FUNCTION_BLOCK FB_FormingBoardControl_V1
VAR_INPUT
    // ── Group / Interlocks ───────────────────────────────────────────────────────
    startGroup                   : BOOL;   // Start command (pulse / rising edge)
    stopGroup                    : BOOL;   // Stop command  (pressed / level)
    groupReset                   : BOOL;   // Group fault Reset (Comando reset falhas do grupo)

    // ── VFD per-drive status inputs ─────────────────────────────────────────────
    formingBoardTractionRollFault               : BOOL;   // VFD ready/healthy (master)
	formingBoardTractionRollCoolingFault  : BOOL;   // VFD ready/healthy (master)
    formingBoardTractionRollVfdRunFeedback         : BOOL;   // VFD RUN feedback  (master)
    formingBoardTractionRollVfdFaultFeedback       : BOOL;   // VFD fault         (master)
   
	formingBoardSuctionRollFault                : BOOL;   // VFD ready/healthy (slave)
	formingBoardSuctionRollCoolingFault		: BOOL;   // VFD ready/healthy (slave)	
	
    formingBoardSuctionVfdRunFeedback          : BOOL;   // VFD RUN feedback  (slave)
    formingBoardSuctionVfdFaultFeedback        : BOOL;   // VFD fault         (slave)

    // ── Speed Setpoints ─────────────────────────────────────────────────────────
    groupAutoSpeedMPM            : REAL;   // Auto speed setpoint [m/min]
    groupMaxSpeed                : REAL := 600.0; // Max allowed line speed [m/min]

    // ── Auto / Manual ───────────────────────────────────────────────────────────
    groupSpeedAutoMan            : BOOL;   // 0=Manual / 1=Auto
    groupManualSpeedMPM          : REAL := 50.0;  // Manual speed [m/min]

    // ── Feedbacks ───────────────────────────────────────────────────────────────
    masterTorqueFeedback         : REAL;   // [% or Nm]
    slaveTorqueFeedback          : REAL;   // [% or Nm]
    masterSpeedFeedback          : REAL;   // [m/min or %] — be consistent
    slaveSpeedFeedback           : REAL;   // [m/min or %] — be consistent

    // ── Ratio & Offsets ─────────────────────────────────────────────────────────
    masterSlaveGearRatio		: REAL := 1.0;   // Slave/Master speed ratio
// 	interGroupGearRatio			: REAL := 1.0;   // Speed diference btween groups
	
    slaveTorqueOfsset            : REAL := 0.0;   // (typo kept) torque trim [%/Nm]
    slaveSpeedOffset             : REAL := 10;    // Offset as % of master speed (+5 => +5%)

    // ── Torque control parameters ───────────────────────────────────────────────
    torqueLimitMinPct            : REAL := 5.0;   // Min torque [%]  (allow negative if regen)
    torqueLimitMaxPct            : REAL := 100.0; // Max torque [%]
    torqueDeadbandPct            : REAL := 1.0;   // |torque| below => 0 (noise cleanup)
	
    torqueFilterTime             : TIME := T#1MS;
    displayFilterTime             : TIME := T#20MS;	

    // ── Dynamics (for ramp block) ───────────────────────────────────────────────
    rampRate                     : REAL := 0.01;  // Ref accel mag in %/s (A_UP=+rampRate, A_DN=-rampRate)

    // ── Speed difference limit ──────────────────────────────────────────────────
    speedDiferenceLimit          : REAL := 5.0;
	
	
	
	
	//Headbox inputs
	
	//==============================================================
	// FORMING BOARD — WIRE EDGE OVERRUN SENSORS
	//==============================================================
	formingBoardWireOverrunOperatorSideSensor : BOOL;  // TRUE when wire overruns on operator side
	formingBoardWireOverrunDriveSideSensor    : BOOL;  // TRUE when wire overruns on drive/motor side	

	//==============================================================
	// HEADBOX LIPS OPENING CONTROL — VARIABLES
	//==============================================================
	
	// Position feedback and physical limits [mm]
	headboxLipsPositionFeedback_mm     : REAL;          // Actual lips opening [mm]
	headboxLipsMinOpening_mm           : REAL := 0.0;   // Minimum allowed opening [mm]
	headboxLipsMaxOpening_mm           : REAL := 25.0;  // Maximum allowed opening [mm]
	
	// Limit sensors (digital inputs)
	headboxLipsLimitFullyOpen          : BOOL;          // TRUE when fully open (max) limit sensor active
	headboxLipsLimitFullyClosed        : BOOL;          // TRUE when fully closed (min) limit sensor active
	
	// Manual jog commands (for manual mode)
	headboxLipsManualOpenCmd           : BOOL;          // Jog open while pressed
	headboxLipsManualCloseCmd          : BOOL;          // Jog close while pressed
	
	// Automatic positioning (for auto mode)
	headboxLipsTargetSetpoint_mm       : REAL;          // Desired lips opening [mm]
	headboxLipsAutoAdjustCmd           : BOOL;          // Pulse to start auto adjustment
	
		
	formingBoardRollUpCmd        : BOOL;  // Command to move forming board UP (active-high)
	formingBoardRollDownCmd      : BOOL;  // Command to move forming board DOWN (active-high)
	formingBoardRollLimitUpSensor    : BOOL;  // TRUE when upper limit is reached (prevents further UP)
	formingBoardRollLimitDownSensor  : BOOL;  // TRUE when lower limit is reached (prevents further DOWN)
	formingBoardRollUpDownMotorFault            : BOOL;  // TRUE = fault present → disables all movement	
	
	formingBoardStretchCmd           : BOOL;  // Jog command to stretch (increase tension)
	formingBoardUnstretchCmd         : BOOL;  // Jog command to unstretch (decrease tension)
	formingBoardLimitStretchSensor   : BOOL;  // TRUE when maximum stretch limit is reached
	formingBoardLimitUnstretchSensor : BOOL;  // TRUE when minimum stretch limit is reached
	formingBoardStretchMotorFault         : BOOL;  // Fault interlock for stretch unit
	
		
END_VAR

VAR_OUTPUT
    deviceState                  : STRING;
    groupFault                   : BOOL;   // Fault present (Falha do grupo)

    // ── Drive References (0..100%) ──────────────────────────────────────────────
    masterDriveSpeedRefPct       : REAL;   // Master reference [%]
    slaveDriveSpeedRefPct        : REAL;   // Slave  reference [%]
	nextGroupSpeedRefPct		 : REAL;   // Next group reference [%]
	nextGroupSpeedRefMPM		 : REAL;   // Next group reference [Meters per minute]
	
    // ── Torque limit to slave (from master torque path / or PID) ───────────────
    slaveDriveTorqueLimit        : REAL;   // [% or Nm]

    // ── Drive Commands ──────────────────────────────────────────────────────────
    masterDriveEnable            : BOOL;
    slaveDriveEnable             : BOOL;
    masterDriveReset             : BOOL;
    slaveDriveReset              : BOOL;

    // ── Diagnostics ─────────────────────────────────────────────────────────────
    currentSpeedDifence          : REAL;

    // ── Group status & HMI displays ────────────────────────────────────────────
    statusCode                   	: INT;    // 0=Idle, 1=Starting, 2=Running, 3=Fault (group)
	
    masterSpeedMPMFilteredDisplay   : REAL;   // Filtered master speed [m/min]
    slaveSpeedMPMFilteredDisplay    : REAL;   // Filtered slave  speed [m/min]
	
    masterTorqueFilteredDisplay  	: REAL;   // Master torque (raw)  [% or Nm]
    slaveTorqueFilteredDisplay   	: REAL;   // Slave torque (filtered) [% or Nm]

    // ── NEW: per-drive motor status codes ───────────────────────────────────────
    masterStatusCode             : INT;    // 0=Idle, 1=Starting, 2=Running, 3=Fault
    slaveStatusCode              : INT;    // 0=Idle, 1=Starting, 2=Running, 3=Fault
	
	//==============================================================
	// HEADBOX LIPS OPENING CONTROL — OUTPUTS
	//==============================================================
	
	// Drive outputs (modulated by PWM in automatic mode)
	headboxLipsOpenCmd                : BOOL;  // Output to open lips (PWM-modulated in Auto mode)
	headboxLipsCloseCmd               : BOOL;  // Output to close lips (PWM-modulated in Auto mode)
	headboxLipsPosition_mm       		  : REAL;  // Target − Feedback error [mm]
	
	//==============================================================
	// FORMING BOARD — ROLL DRIVE OUTPUTS
	//==============================================================
	formingBoardRollUp       : BOOL;  // Output to drive the forming board UP
	formingBoardRollDown     : BOOL;  // Output to drive the forming board DOWN
	
	//==============================================================
	// FORMING BOARD — STRETCH DRIVE OUTPUTS
	//==============================================================
	formingBoardStretch      : BOOL;  // Output to stretch (increase tension)
	formingBoardUnstretch    : BOOL;  // Output to unstretch (decrease tension)
		

	hmiAlarms 				: PaperMachine_TypeHmiAlarms; 	

END_VAR

VAR
    // ── Internals / Ramps ───────────────────────────────────────────────────────
    rampTargetPct                : REAL;   // 0..100% target into ramp
    instFB_Gen_SRamp             : FB_Gen_SRamp; // Your ramp FB

    // ── State & Edges ───────────────────────────────────────────────────────────
    state                        : INT;    // 0=IDLE,1=ENABLE,2=WAIT_EN,3=RAMP_EN,4=RUN,5=STOPPING,10=FAULT
    startGroupOld                : BOOL;
    stopGroupOld                 : BOOL;
    rStart                       : BOOL;
    rStop                        : BOOL;

    // ── Timers & thresholds ─────────────────────────────────────────────────────
    instTONEnableWait            : TON;
    instTONStopWait              : TON;
    enableTimeout                : TIME := T#5s;  // Wait for op-enable
    stopTimeout                  : TIME := T#8s;  // Max wait to speed≈0
    speedZeroThresholdPct        : REAL := 4.00;  // Consider stopped if |speed| ≤ this
    epsRefPct                    : REAL := 0.05;  // Small epsilon for ref≈0

    // ── Ramp control ────────────────────────────────────────────────────────────
    rampReset                    : BOOL;   // Resets ramp (sets Y/V to 0 in your FB)

    // ── Filter state used by _TorqueReference ───────────────────────────────────
    torqueFiltY                  : REAL;   // last filtered torque
    torqueFiltInit               : BOOL;   // init flag (bumpless start)
    instsFT_PT1TorqueFilter      : FT_PT1;

    // ── Speed difference supervision ────────────────────────────────────────────
    instTONSpeedDifDelay         : TON;

    // ── HMI-only PT1 filters ───────────────────────────────────────────────────
    instPT1_MasterSpeedDisplay          : FT_PT1;
    instPT1_SlaveSpeedDisplay           : FT_PT1;
	
    instPT1_MasterTorqueDisplay  		: FT_PT1;
    instPT1_SlaveTorqueDisplay   		: FT_PT1;
	
	instFB_HeadboxLipsPWMControl		: FB_HeadboxLipsPWMControl;	
	
END_VAR

// ─────────────────────────────────────────────────────────────────────────────
// MAIN CALL SEQUENCE
// ─────────────────────────────────────────────────────────────────────────────
_FeedbackDisplay();
_GroupControl();          // 1) State machine: edges, enables, stop modes
_ReferenceGenerator();    // 2) Build master/slave references with ramp
_TorqueReference();       // 3) Legacy torque transfer (kept)
_StateDisplay();

_SpeedDifferenceCheck();  // 4) Speed difference monitor & trip
_headboxLipsPosition();

_auxiliaryControls();
_alarmsDisplay();

METHOD _alarmsDisplay
VAR_INPUT
END_VAR
//==============================================================
// FAULT EVALUATION — PER CONDITION (flags only; no global set)
//==============================================================

//----------------------------
// FORMING BOARD DRIVES
//----------------------------
hmiAlarms.formingBoardRollDriveFaultAlarm    := formingBoardRollUpDownMotorFault;
hmiAlarms.formingBoardStretchDriveFaultAlarm := formingBoardStretchMotorFault;

//----------------------------
// FORMING BOARD AUXILIARY MOTORS
//----------------------------
hmiAlarms.formingBoardSuctionRollFaultAlarm         := formingBoardSuctionRollFault;
hmiAlarms.formingBoardSuctionRollCoolingFaultAlarm  := formingBoardSuctionRollCoolingFault;
hmiAlarms.formingBoardTractionRollFaultAlarm        := formingBoardTractionRollFault;
hmiAlarms.formingBoardTractionRollCoolingFaultAlarm := formingBoardTractionRollCoolingFault;

//----------------------------
// FORMING BOARD WIRE OVERRUN
//----------------------------
hmiAlarms.formingBoardWireOverrunOperatorSideAlarm := formingBoardWireOverrunOperatorSideSensor;
hmiAlarms.formingBoardWireOverrunDriveSideAlarm    := formingBoardWireOverrunDriveSideSensor;

//----------------------------
// FORMING BOARD GROUP FAULT STATUS
//----------------------------
groupFault :=
    hmiAlarms.formingBoardRollDriveFaultAlarm OR
    hmiAlarms.formingBoardStretchDriveFaultAlarm OR
    hmiAlarms.formingBoardSuctionRollFaultAlarm OR
    hmiAlarms.formingBoardSuctionRollCoolingFaultAlarm OR
    hmiAlarms.formingBoardTractionRollFaultAlarm OR
    hmiAlarms.formingBoardTractionRollCoolingFaultAlarm OR
    hmiAlarms.formingBoardWireOverrunOperatorSideAlarm OR
    hmiAlarms.formingBoardWireOverrunDriveSideAlarm;
END_METHOD

METHOD _auxiliaryControls
VAR_INPUT
END_VAR
//============================
// FORMING BOARD ROLL UP/DOWN
//============================
IF NOT formingBoardRollUpDownMotorFault THEN
    IF formingBoardRollUpCmd AND NOT formingBoardRollDownCmd AND NOT formingBoardRollLimitUpSensor THEN
        formingBoardRollUp := TRUE;
    ELSE
        formingBoardRollUp := FALSE;
    END_IF;

    IF formingBoardRollDownCmd AND NOT formingBoardRollUpCmd AND NOT formingBoardRollLimitDownSensor THEN
        formingBoardRollDown := TRUE;
    ELSE
        formingBoardRollDown := FALSE;
    END_IF;
ELSE
    formingBoardRollUp := FALSE;
    formingBoardRollDown := FALSE;
END_IF;


//============================
// FORMING BOARD STRETCH/UNSTRETCH
//============================
IF NOT formingBoardStretchMotorFault THEN
    IF formingBoardStretchCmd AND NOT formingBoardUnstretchCmd AND NOT formingBoardLimitStretchSensor THEN
        formingBoardStretch := TRUE;
    ELSE
        formingBoardStretch := FALSE;
    END_IF;

    IF formingBoardUnstretchCmd AND NOT formingBoardStretchCmd AND NOT formingBoardLimitUnstretchSensor THEN
        formingBoardUnstretch := TRUE;
    ELSE
        formingBoardUnstretch := FALSE;
    END_IF;
ELSE
    formingBoardStretch := FALSE;
    formingBoardUnstretch := FALSE;
END_IF;
END_METHOD

METHOD _FeedbackDisplay
VAR_INPUT
END_VAR
// 5) HMI DISPLAY SIGNALS (filtered speeds/torques + GROUP status)
instPT1_MasterSpeedDisplay(in := masterSpeedFeedback, T := displayFilterTime, K := 1.0, out => masterSpeedMPMFilteredDisplay);
instPT1_SlaveSpeedDisplay (in := slaveSpeedFeedback , T := displayFilterTime, K := 1.0, out => slaveSpeedMPMFilteredDisplay);

instPT1_MasterTorqueDisplay(in := masterTorqueFeedback, T := displayFilterTime, K := 1.0, out => masterTorqueFilteredDisplay);
instPT1_SlaveTorqueDisplay (in := slaveTorqueFeedback , T := displayFilterTime, K := 1.0, out => slaveTorqueFilteredDisplay);
END_METHOD

// ============================== Methods ==============================
// 1) GROUP CONTROL
METHOD _GroupControl
VAR_INPUT
END_VAR
VAR
    speedsNearZero : BOOL;
    refNearZero    : BOOL;
    bothOpEnabled  : BOOL;
END_VAR
// Edges
rStart := startGroup AND NOT startGroupOld;     // Start on pulse
rStop  := stopGroup  AND NOT stopGroupOld;      // Stop also has an edge
startGroupOld := startGroup;
stopGroupOld  := stopGroup;

// Feedback conditions (unit matches your % references)
speedsNearZero :=
    (ABS(masterSpeedFeedback) <= speedZeroThresholdPct) AND
    (ABS(slaveSpeedFeedback)  <= speedZeroThresholdPct);

// Also consider the reference near zero (backup)
refNearZero := ABS(masterDriveSpeedRefPct) <= epsRefPct;

// Use the original "operation enabled" for RUN readiness
bothOpEnabled := formingBoardTractionRollFault AND formingBoardSuctionRollFault;

CASE state OF
    0: // IDLE
        deviceState := 'IDLE';
        rampReset := TRUE;
        IF rStart AND NOT groupFault THEN
            state := 1;
        END_IF

    1: // ENABLE DRIVES
        deviceState := 'ENABLE_DRIVES';
        masterDriveEnable := TRUE;
        slaveDriveEnable  := TRUE;
        rampReset         := TRUE;

        instTONEnableWait(IN := TRUE, PT := enableTimeout);
        IF stopGroup THEN
            instTONEnableWait(IN := FALSE);
            state := 5;
        ELSE
            state := 2;
        END_IF

    2: // WAIT ENABLE FEEDBACK
        deviceState := 'WAIT_ENABLE_FEEDBACK';
        masterDriveEnable := TRUE;
        slaveDriveEnable  := TRUE;
        rampReset         := TRUE;

        instTONEnableWait(IN := TRUE, PT := enableTimeout);

        IF groupFault THEN
            instTONEnableWait(IN := FALSE);
            state := 10;
        ELSIF rStop OR stopGroup THEN
            instTONEnableWait(IN := FALSE);
            state := 5;
        ELSIF bothOpEnabled THEN
            instTONEnableWait(IN := FALSE);
            state := 3;
        ELSIF instTONEnableWait.Q THEN
            instTONEnableWait(IN := FALSE);
            state := 10; // fault: no enable feedback
        END_IF

    3: // RAMP ENABLE (single-cycle gate)
        deviceState := 'RAMP_ENABLE';
        masterDriveEnable := TRUE;
        slaveDriveEnable  := TRUE;
        rampReset         := FALSE; // release ramp now
        IF stopGroup THEN
            state := 5;
        ELSE
            state := 4;
        END_IF

    4: // RUN
        deviceState := SEL(groupSpeedAutoMan,'RUN (Manual)', 'RUN (Auto)');
        masterDriveEnable := TRUE;
        slaveDriveEnable  := TRUE;
        rampReset         := FALSE;

        IF groupFault THEN
            state := 10;
        ELSIF rStop OR stopGroup THEN
            state := 5;
        END_IF

    5: // STOPPING (controlled)
        deviceState := 'STOPPING';
        masterDriveEnable := TRUE;    // keep enabled during decel
        slaveDriveEnable  := TRUE;
        rampReset         := FALSE;   // ramp down references
        // instTONStopWait(IN := TRUE, PT := stopTimeout);  // optional timeout

        // Disable when speed≈0 AND reference≈0
        IF groupFault THEN
            instTONStopWait(IN := FALSE);
            state := 10;

        ELSIF speedsNearZero AND refNearZero THEN
            masterDriveEnable := FALSE;
            slaveDriveEnable  := FALSE;
            instTONStopWait(IN := FALSE);
            state := 0;

        ELSIF instTONStopWait.Q THEN
            masterDriveEnable := FALSE;
            slaveDriveEnable  := FALSE;
            instTONStopWait(IN := FALSE);
            state := 10;
        END_IF

    10: // FAULT
        deviceState := 'FAULT';
        rampReset         := TRUE;    // force ramp outputs to zero
        masterDriveEnable := FALSE;
        slaveDriveEnable  := FALSE;

        // Clear fault when fault disappears and start is low
        IF (NOT groupFault) AND (NOT startGroup) THEN
            state := 0;
        END_IF
END_CASE;
END_METHOD

METHOD _headboxLipsPosition
VAR_INPUT
END_VAR
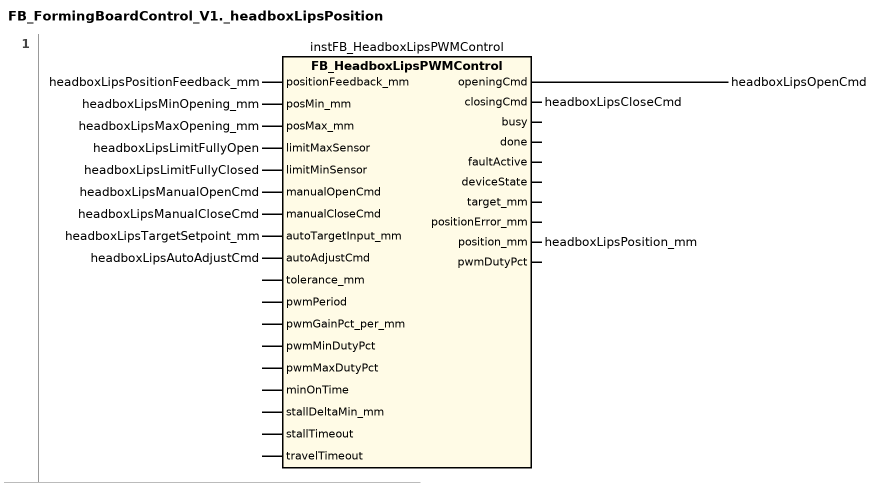
// NETWORK 1
instFB_HeadboxLipsPWMControl(
    positionFeedback_mm := headboxLipsPositionFeedback_mm,
    posMin_mm := headboxLipsMinOpening_mm,
    posMax_mm := headboxLipsMaxOpening_mm,
    limitMaxSensor := headboxLipsLimitFullyOpen,
    limitMinSensor := headboxLipsLimitFullyClosed,
    manualOpenCmd := headboxLipsManualOpenCmd,
    manualCloseCmd := headboxLipsManualCloseCmd,
    autoTargetInput_mm := headboxLipsTargetSetpoint_mm,
    autoAdjustCmd := headboxLipsAutoAdjustCmd,
    closingCmd => headboxLipsCloseCmd,
    position_mm => headboxLipsPosition_mm); // FB_HeadboxLipsPWMControl
headboxLipsOpenCmd := instFB_HeadboxLipsPWMControl.openingCmd;
END_METHOD

// 2) REFERENCE GENERATOR
METHOD _ReferenceGenerator
VAR
    headroomEpsPct      : REAL := 0.20;   // anti-chatter near 100%
    offsetPct           : REAL;
    denom               : REAL;
    maxMasterBySlave    : REAL;
    allowedCapPct       : REAL;
    currMasterPct       : REAL;
    currSlavePct        : REAL;
    targetPct           : REAL;
    cmdSpeedMPM         : REAL;
END_VAR
// 1) Select Auto/Manual command (MPM)
IF groupSpeedAutoMan THEN
    cmdSpeedMPM := groupAutoSpeedMPM;
ELSE
    cmdSpeedMPM := groupManualSpeedMPM;
END_IF

// 2) Scale to 0..100% for the drives
targetPct := _Scale(
    X    := cmdSpeedMPM,
    I_LO := 0.0,          I_HI := groupMaxSpeed,
    O_LO := 0.0,          O_HI := 100.0);

// 3) During STOPPING/FAULT we want zero target; in STOPPING we still ramp down
IF state = 5 THEN
    rampTargetPct := 0.0;
ELSE
    rampTargetPct := targetPct;
END_IF

// --- Pre-limit so SLAVE can’t exceed 100% for given gear + offset ---
offsetPct := slaveSpeedOffset * 0.01;
denom     := masterSlaveGearRatio + offsetPct;

// If denom <= 0, fall back to 100% (no additional cap required)
IF denom > 0.0 THEN
    maxMasterBySlave := 100.0 / denom;   // master % that makes slave hit 100%
ELSE
    maxMasterBySlave := 100.0;
END_IF;

// The cap the master target must obey (also respect master’s own 100%)
allowedCapPct := MIN(100.0, maxMasterBySlave);

// Apply cap to upward commands only (don’t block decel)
rampTargetPct := MIN(rampTargetPct, allowedCapPct);

// --- Freeze upward if currently at/near limit (anti-overrun using current refs) ---
currMasterPct := instFB_Gen_SRamp.Y;                          // current master ref (%)
currSlavePct  := LIMIT(0.0, currMasterPct * (masterSlaveGearRatio + offsetPct), 100.0);

IF (currMasterPct >= 100.0 - headroomEpsPct) OR
   (currSlavePct  >= 100.0 - headroomEpsPct) THEN
    // Prevent increasing the target above current value; allow decreases
    rampTargetPct := MIN(rampTargetPct, currMasterPct);
END_IF

// 4) Ramp call (unchanged)
instFB_Gen_SRamp(
    X          := rampTargetPct,
    A_UP       := MAX(0.0, rampRate),
    A_DN       := -MAX(0.0, rampRate),
    VU_MAX     := 1000.0,
    VD_MAX     := -1000.0,
    LIMIT_HIGH := 100.0,
    RST        := rampReset);

IF state = 5 THEN
    instFB_Gen_SRamp.LIMIT_LOW := 0.0;
ELSE
    instFB_Gen_SRamp.LIMIT_LOW := 3.5;
END_IF

// 5) Master reference = ramp Y but also respect the slave-driven cap
masterDriveSpeedRefPct := MIN(instFB_Gen_SRamp.Y, allowedCapPct);

// 6) Slave reference: gear + offset, then clamp 0..100
slaveDriveSpeedRefPct :=
    LIMIT(0.0, masterDriveSpeedRefPct * (masterSlaveGearRatio + offsetPct), 100.0);

// 7) Final safety clamp for master (symmetry) + forward as % to next group
masterDriveSpeedRefPct := LIMIT(0.0, masterDriveSpeedRefPct, 100.0);
nextGroupSpeedRefPct   := masterDriveSpeedRefPct;

// 8) Also forward the next group reference in MPM (easy to replicate elsewhere)
nextGroupSpeedRefMPM := _Scale(
    X    := nextGroupSpeedRefPct,
    I_LO := 0.0,          I_HI := 100.0,
    O_LO := 0.0,          O_HI := groupMaxSpeed);
END_METHOD

METHOD PRIVATE _Scale : REAL
VAR_INPUT
    X    : REAL;
    I_LO : REAL;
    I_HI : REAL;
    O_LO : REAL;
    O_HI : REAL;
END_VAR
IF I_LO = I_HI THEN
	_Scale := O_LO;
ELSE
	_Scale := (O_HI - O_LO) / (I_HI - I_LO) * (LIMIT(I_LO, X, I_HI) - I_LO) + O_LO;
END_IF;
END_METHOD

// 6) OPTIONAL: SLAVE TORQUE PID TRACKING (new)
METHOD _SlaveTorquePID
VAR_INPUT
    enablePID : BOOL := TRUE;   // TRUE=PID active, FALSE=hold/track current output
    Kp        : REAL := 0.8;    // proportional gain (tune as needed)
    Tn        : REAL := 1.5;    // integral time [s]
    Tv        : REAL := 0.0;    // derivative time [s]
END_VAR
VAR
    masterFilt : REAL;
    slaveFilt  : REAL;
    sp         : REAL;  // setpoint (master)
    pv         : REAL;  // process value (slave)
    y          : REAL;  // PID output (pre-clamp)
    e          : REAL;  // SET - ACT (diagnostic)
    limMin     : REAL;
    limMax     : REAL;
END_VAR
VAR_STAT
    pid        : CTRL_PID;  // PID instance (retained)
    fMaster    : FT_PT1;    // PT1 for master torque
    fSlave     : FT_PT1;    // PT1 for slave torque
END_VAR
// 1) Filter master & slave torques (reuse existing time constant)
fMaster(in := masterTorqueFeedback, T := torqueFilterTime, K := 1.0, out => masterFilt);
fSlave (in := slaveTorqueFeedback , T := torqueFilterTime, K := 1.0, out => slaveFilt);

// 2) Build setpoint and PV
sp := masterFilt + slaveTorqueOfsset;   // follow master + configured trim
pv := slaveFilt;

// 3) Limits from existing configuration
limMin := torqueLimitMinPct;
limMax := torqueLimitMaxPct;

// 4) PID with bumpless transfer (manual input tracks current output when disabled)
pid(
    ACT := pv,                      // process value (slave torque)
    SET := sp,                      // setpoint (master torque)
    MAN := NOT enablePID,           // MAN=TRUE => manual/track
    M_I := slaveDriveTorqueLimit,   // track current output for bumpless re-enable
    RST := FALSE,                   // external reset (unused)
    KP  := Kp,
    TN  := Tn,
    TV  := Tv,
    LL  := limMin,
    LH  := limMax,
    Y   => y,
    DIFF=> e,
    LIM =>                          // unused
);

// 5) Clamp and publish
slaveDriveTorqueLimit := LIMIT(limMin, y, limMax);
END_METHOD

METHOD PRIVATE _SpeedDifferenceCheck
VAR
    diff : REAL;
END_VAR
// 1) Absolute difference Master-Slave
diff := ABS(masterSpeedMPMFilteredDisplay - slaveSpeedMPMFilteredDisplay);
currentSpeedDifence := diff;

// 2) If beyond limit -> stop group (with a small delay)
IF diff > speedDiferenceLimit THEN
    instTONSpeedDifDelay.IN := TRUE;
    instTONSpeedDifDelay.PT := T#2S;

    IF instTONSpeedDifDelay.Q THEN
        state := 10;                  // Fault
        deviceState := 'FAULT: Speed difference exceeded';
    END_IF
ELSE
    instTONSpeedDifDelay.IN := FALSE;
END_IF

instTONSpeedDifDelay();
END_METHOD

METHOD _StateDisplay
VAR_INPUT
END_VAR

// ──────────────────────────────────────────────────────────────────────────────
// _StateDisplay
// Maps the internal machine "state" to a compact HMI status code and derives
// per-drive motor status codes from VFD signals.
//
// statusCode / masterStatusCode / slaveStatusCode legend:
//   0 = Idle, 1 = Starting, 2 = Running, 3 = Fault
//
// Machine "state" groups:
//   0 = IDLE, 1 = ENABLE, 2 = WAIT_EN, 3 = RAMP_EN, 4 = RUN, 5 = STOPPING, 10 = FAULT
// Priority rule (for motors): Fault > Running > Starting > Idle
// ──────────────────────────────────────────────────────────────────────────────
VAR CONSTANT
    STATUS_IDLE     : INT := 0;
//    STATUS_STARTING : INT := 1;
    STATUS_RUNNING  : INT := 1;
    STATUS_FAULT    : INT := 2;
END_VAR

// ─────────────── Group machine states into a single HMI statusCode ───────────
CASE state OF
    10: // FAULT
        statusCode := STATUS_FAULT;

    4:  // RUN
        statusCode := STATUS_RUNNING;

    1, 2, 3: // ENABLE / WAIT_EN / RAMP_EN
//        statusCode := STATUS_STARTING;

    ELSE // IDLE, STOPPING, or any other unlisted state
        statusCode := STATUS_IDLE;
END_CASE;

// ─────────────── Helper pattern for per-drive status (inline) ────────────────
// Evaluation order enforces priority: Fault > Running > Starting > Idle

// Master drive
IF formingBoardTractionRollVfdFaultFeedback THEN
    masterStatusCode := STATUS_FAULT;
ELSIF formingBoardTractionRollVfdRunFeedback THEN
    masterStatusCode := STATUS_RUNNING;
ELSE
    masterStatusCode := STATUS_IDLE;
END_IF;

// Slave drive
IF formingBoardSuctionVfdFaultFeedback THEN
    slaveStatusCode := STATUS_FAULT;
ELSIF formingBoardSuctionVfdRunFeedback THEN
    slaveStatusCode := STATUS_RUNNING;
ELSE
    slaveStatusCode := STATUS_IDLE;
END_IF;
END_METHOD

METHOD _TorqueReference
VAR
    rawTorque     : REAL;
    filtTorque    : REAL;
    torqueCmd     : REAL;
    limitedTorque : REAL;
    clamped       : BOOL;
END_VAR
// 1) Read master torque (keep units consistent with your limits)
rawTorque := masterTorqueFeedback;

// 2) Low-pass filter (OSCAT PT1)
instsFT_PT1TorqueFilter(
    in  := rawTorque,
    T   := torqueFilterTime,   // time constant in seconds (e.g., 0.25)
    K   := 0.8,                // unity gain
    out => filtTorque
);

// 3) Deadband cleanup
IF ABS(filtTorque) < torqueDeadbandPct THEN
    filtTorque := 0.0;
END_IF

// 4) Apply offset between master and slave
torqueCmd := filtTorque + slaveTorqueOfsset;

// 5) Clamp to limits
limitedTorque := LIMIT(torqueLimitMinPct, torqueCmd, torqueLimitMaxPct);
clamped       := (limitedTorque <> torqueCmd);

// 6) Output
slaveDriveTorqueLimit := limitedTorque;


//slaveDriveTorqueLimit := LIMIT(torqueLimitMinPct, masterTorqueFeedback, torqueLimitMaxPct);
END_METHOD

END_FUNCTION_BLOCK

(* stored: Version 1.1.0.1, ProductVersion 3.1.4024.15
   POU FB_FormingBoardControl_V1: Id {0341cbdf-b8a3-4b8d-9801-cb7e35cafbf7}, SpecialFunc None
   Method _alarmsDisplay: Id {0461d554-8be0-4155-a22f-684dbe18fcea}
   Method _auxiliaryControls: Id {a22de1c9-6b9a-4972-be03-0a4d0f8183e9}
   Method _FeedbackDisplay: Id {9787b19e-cb2a-4ad6-b3b8-527a44a0dd75}
   Method _GroupControl: Id {ffb736eb-8f73-4dad-91a7-f4ecebade366}
   Method _headboxLipsPosition: Id {ae440f30-7006-4b9b-8786-c39621402025}
   Method _ReferenceGenerator: Id {d1bebbfa-bfe1-4125-b9cf-abcf61a22a04}
   Method _Scale: Id {70e52522-893d-4230-ac46-b736c1d79a1d}
   Method _SlaveTorquePID: Id {d2f2c034-a009-466c-a7c6-a830587846dc}
   Method _SpeedDifferenceCheck: Id {04e52e61-860d-4025-9001-97f886bc892a}
   Method _StateDisplay: Id {d53a5fea-f9d1-4630-b78f-0baae473f501}
   Method _TorqueReference: Id {1898f17f-1d1c-48e9-86d0-81f7e5611d7a} *)
